PROGRAM EVACUAZIONE_SCARTI
VAR

	bINIT					:BOOL;
	
	//act Area MACINATORE
	rtAuto_ON				:R_TRIG;
	ftAuto_ON				:F_TRIG;
	tmrT3_ON				:TON;	
	tmrT3_OFF				:TON;		
	tmrT1T2_ON				:TON;	
	tmrT1T2_OFF				:TON;
	ft_AbilitaT1T2			:F_TRIG;
	ft_AbilitaT3			:F_TRIG;
	ft_AbilitaT4			:F_TRIG;
	
	Area_HS_On				:BOOL;
	rt_Area_M_Riarmo		:R_TRIG;
	rt_Area_M_Disarmo		:R_TRIG;
	tmr_SvuotaT1			:TON;		
	tmr_SvuotaT2			:TON;	
	tmr_SvuotaT3			:TON;	
	tmr_MacinatoreON		:TON;
	tmr_MacinatoreOFF		:TON;
	rt_MacinatoreON			:R_TRIG;
	rt_MacinatoreOFF		:R_TRIG;
	rt_MPO1_btn_M_MacOn		:R_TRIG;
	rt_btn_Fsx_T3StartMan	:R_TRIG;
	rt_btn_Fdx_T4StartMan	:R_TRIG;
	tmr_T3T5T6DelayStart	:TON;
	rt_T3S1full				:R_TRIG;
	tmr_T3S1vuoto			:TON;
	tmr_T3S1pieno			:TON;
	bT3S1full				:BOOL;
	rt_T3S2full				:R_TRIG;
	tmr_T3S2vuoto			:TON;
	bT3S2full				:BOOL;
	ft_T3S2full				:F_TRIG;
	countT3avanzamento		:INT;
	
	//act AREA SILOS
	rt_Area_S_Riarmo		:R_TRIG;
	rt_Area_S_Disarmo		:R_TRIG;
	
	//act_ALARM
	rtAlarmReset			:R_TRIG;	
	AlarmActive				:BOOL;
	AlarmReset				:BOOL;
	AlarmMask				:DWORD;
	T5_Bloccato				:ES_ALARM;	
	T6_Bloccato				:ES_ALARM;
	tmr_T4ON				:TON;
	
	tmrT3_Lavoro			:TON;	
	tmrT3_Pausa				:TON;
	tmrT5T6_RitStop			:TOF;	
	tmrS1_T_Rit_Empty		:TOF;
	tmrT1S01_Full			:TON;
	tmr_T_Rit_Stop_T4T5T6	:TOF;
	
	Forza_TT1S01_Full		:BOOL;
	
	appT1S01_Full			: BOOL;
	
	En_T_RitStopT5T6		:BOOL;
	
	//SENSORI	
	S1						:ES_S1;
	S2						:ES_S2;
	T1						:ES_T1;
	T3						:ES_T3;
	T5						:ES_T5;
	T6						:ES_T6;
                        	
	T1SO1tmravg				:TON;
	T1SO1arravg				:ARRAY[0..99]OF INT;
	T1SO1maxCnt				:INT;
	T1SO1sumavg				:REAL;
	T1SO1avg				:REAL;
	T1SO1cnt				:INT;
	T1SO1cnt2				:INT;	
	T1SO1cnt3				:INT;
	                    	
	S1SO2tmravg				:TON;
	S1SO2arravg				:ARRAY[0..99]OF INT;
	S1SO2maxCnt				:INT;
	S1SO2sumavg				:REAL;
	S1SO2avg				:REAL;
	S1SO2cnt				:INT;
	S1SO2cnt2				:INT;	
	S1SO2cnt3				:INT;		
                        	
	T3S1tmravg				:TON;
	T3S1arravg				:ARRAY[0..99]OF INT;
	T3S1maxCnt				:INT;
	T3S1sumavg				:REAL;
	T3S1avg					:REAL;
	T3S1cnt					:INT;
	T3S1cnt2				:INT;	
	T3S1cnt3				:INT;
	                    	
	T3S2tmravg				:TON;
	T3S2arravg				:ARRAY[0..99]OF INT;
	T3S2maxCnt				:INT;
	T3S2sumavg				:REAL;
	T3S2avg					:REAL;
	T3S2cnt					:INT;
	T3S2cnt2				:INT;	
	T3S2cnt3				:INT;
	                    	
	//SEMAFORI          	
	fbS1_Se1				:FB_Semaforo;
		
	//gestione filtro temporale sensore 
	SO2_full_curr			:BOOL;
	tmrValidaSoglia_S02		:TON;

	
	//gestione macinatore
	TON_Macinatore_On			:TON;
	TON_Vibro_Macinatore_On		:TON;
	TON_Ciclo_Macinatore		:TON;
	TP_Start_Macinatore			:TP;
	TP_Stop_Macinatore			:TP;

	TS							:BOOL;
	M_Ciclo_Svuotamento_Hdd_RUN	:BOOL;
	M_Auto_Start_Macinatore		:BOOL;
	M_Auto_Start_Vibro_Macinatore		:BOOL;
	M_Auto_Start_Vibro_Hdd		:BOOL;
	M_Start_Req_Stop_Macinatore	:BOOL;	
	M_Stop_Req_Stop_Macinatore	:BOOL;
	
	M_Man_Start_Vibro_Hdd		:BOOL;
	
	
	
	
	//TwinsAFE
	tmrErrAck				:TON;	
	
END_VAR
VAR // added by the converter: edge detectors and wires of the graphical bodies
    _rt1, _rt2 : R_TRIG;
    _w1, _w2, _w3 : BOOL;
    _ft1 : F_TRIG;
END_VAR


act_INIT();

act_ALARM();

act_INPUT();

act_Sensori();

act_AreaSilos();

act_Macinatore();

//act_AreaMac_AUTO();
//act_AreaMac_MAN();

act_Semafori();

act_OUTPUT();

act_HMI();

ACTION act_ALARM:

//TwinSAFE
TS_ErrAck := C1P1_Rst_Eme OR R1P1_Rst_Eme;


tmrErrAck(IN:=TS_ErrAck,PT:=T#1S);
IF tmrErrAck.Q THEN
	TS_ErrAck:=FALSE;
END_IF




//ALLARMI DA SENSORI
rtAlarmReset(CLK:=bAlarmReset);
IF rtAlarmReset.Q THEN
	bAlarmReset:=FALSE;
	T5.Alarm.Active:=FALSE;	
	T6.Alarm.Active:=FALSE;	
	bAllarmeT5:=FALSE;
	bAllarmeT6:=FALSE;
END_IF

IF NOT AlarmActive THEN

	//Allarme T5 Bloccato - 5s
	IF HQ1_T5_KA5 THEN
		T5.Alarm.tmr(IN:=TRUE,PT:=INT_TO_TIME(T5.Alarm.pt*1000));
		IF T5.Alarm.tmr.ET < T5.Alarm.tmr.PT THEN
			T5.S1_rt(CLK:=T5_S1);
			IF T5.S1_rt.Q THEN
				T5.S1_letto:=TRUE;		
			END_IF
		END_IF
	
		IF T5.Alarm.tmr.Q THEN
			IF NOT T5.S1_letto AND HQ1_T5_KA5 THEN
				T5.Alarm.Active:=TRUE AND bAllarmeT5enable;	
			ELSE	
				T5.Alarm.Active:=FALSE;	
			END_IF
			T5.S1_letto:=FALSE;
			T5.Alarm.tmr(IN:=FALSE);
		END_IF
	END_IF

	
	
		
	//Allarme T6 Bloccato - 5s
	IF HQ1_T6_KA6 THEN
		T6.Alarm.tmr(IN:=TRUE,PT:=INT_TO_TIME(T6.Alarm.pt*1000));
		IF T6.Alarm.tmr.ET < T6.Alarm.tmr.PT THEN
			T6.S1_rt(CLK:=T6_S1);
			IF T6.S1_rt.Q THEN
				T6.S1_letto:=TRUE;		
			END_IF
		END_IF
	
		IF T6.Alarm.tmr.Q THEN
			IF NOT T6.S1_letto AND HQ1_T6_KA6 THEN
				T6.Alarm.Active:=TRUE AND bAllarmeT6enable;	
			ELSE	
				T6.Alarm.Active:=FALSE;	
			END_IF
			T6.S1_letto:=FALSE;
			T6.Alarm.tmr(IN:=FALSE);
		END_IF	
	END_IF
	

	
	
	//Allarme S2 Silos Pieno
	IF S2.S1_full (*AND glo_ES_BtnHMI.S2_Alarm_Enable*) THEN
		S2.Alarm.Active := TRUE AND bAllarmeS2S1enable;
	END_IF
	
	
	
	
	//Allarme T3 Bloccato - 30s
	IF T1.SO1_full AND T3.S1_full THEN
		T3.Alarm.tmr(IN:=TRUE,PT:=INT_TO_TIME(T3.Alarm.pt*1000));
		IF T3.Alarm.tmr.Q THEN
			T3.Alarm.tmr(IN:=FALSE);
			T3.Alarm.Active := TRUE;	
		END_IF
	ELSE
		T3.Alarm.Active := FALSE;
	END_IF	

	
	
	
	//Allarme S1 Silos1 Pieno
	IF (*S1_S2_full AND*) S1_S2 THEN
		S1.Alarm.Active:=TRUE;
	END_IF
	
END_IF
END_ACTION

ACTION act_AreaMac_AUTO:

//#######################################################
//###################    AREA M ON    ###################
//#######################################################

IF M_PO1.key THEN
	rt_Area_M_Riarmo(CLK:= M_PO1.btn_R_Riarmo OR bSIMULA_btnR);
	IF rt_Area_M_Riarmo.Q THEN
		bSIMULA_btnR:=FALSE;
		AreaM_ON:= TRUE;
	END_IF
END_IF
rt_Area_M_Disarmo(CLK:= M_PO1.btn_0_AreaMoff OR bSIMULA_btn0);
IF NOT M_PO1.key OR rt_Area_M_Disarmo.Q OR NOT TS_AreaM_ON OR NOT TS_AreaS_ON (*OR NOT TS_AreaM_OFF*) THEN
	bSIMULA_btn0:=FALSE;	
	AreaM_ON:=FALSE;
	fun_AreaM_SPEGNITUTTO();	
END_IF

//#######################################################
//##################     AUTOMATICO   ###################
//#######################################################

rtAuto_ON(CLK:=HQ1_Auto_ON OR bSIMULAAuto_ON);
IF rtAuto_ON.Q THEN
	bIsAuto:=TRUE;
END_IF
ftAuto_ON(CLK:=HQ1_Auto_ON OR bSIMULAAuto_ON);
IF ftAuto_ON.Q THEN
	bIsAuto:=FALSE;	
	bSIMULA_btn0:=TRUE;	
	bSIMULA_btn0silos:=TRUE;	
	fun_AreaM_SPEGNITUTTO();	
END_IF

IF bIsAuto THEN
	

	//#######################################################
	//####################     T1 - T2    ###################
	//#######################################################
	
	(*
	- sensore sotto hundegger dà che T1 è pieno
	- area attiva
	- sensore all'inizio del T3 dà che è vuoto/libero
	- T3 non è bloccato: sensori del T1 e T3 contemporaneamente non pieni
	*)
	
	IF bAbilitaT1T2 THEN
		
		CASE stepT1T2 OF
			
			0:
				descT1T2:='T1-T2 spenti. In attesa di T1SO1 pieno';
				IF T1.SO1_full THEN
					stepT1T2:=5;
				END_IF
			
			5:
				IF NOT T3.S1_full (*AND NOT T3.Alarm.Active*) THEN 
					descT1T2:='Avvio T1-T2';
					bT1_ON:=TRUE;
					bT2_ON:=TRUE;
					tmrT1T2_ON(IN:=FALSE);
					stepT1T2:=10;
				ELSIF T3.S1_full (*OR T3.Alarm.Active*) THEN
					stepT1T2:=100;
				END_IF
			
			10:
				descT1T2:='T1-T2 accesi per 2s';
				tmrT1T2_ON(IN:=TRUE,PT:=T#2S);
				IF tmrT1T2_ON.Q THEN
					tmrT1T2_OFF(IN:=FALSE);
					stepT1T2:=15;					
				END_IF
			
			15:
				descT1T2:='T1-T2 accesi finchè T3S1 pieno';		
				IF NOT T1.SO1_full THEN
					tmrT1T2_ON(IN:=FALSE);					
					bT1_ON:=FALSE;
					stepT1T2:=16;
				END_IF		
				tmr_T3S1pieno(in:=T3.S1_full,PT:=T#2S);
				IF tmr_T3S1pieno.Q THEN
					bT1_ON:=FALSE;
					bT2_ON:=FALSE;
					stepT1T2:=20;				
				END_IF
	
			16:
				descT1T2:='T1spento, T2 acceso per 15s o finchè T3S1 pieno';	
				tmrT1T2_ON(IN:=TRUE,PT:=T#15S);	
				IF tmrT1T2_ON.Q OR T3.S1_full THEN
					bT2_ON:=FALSE;
					stepT1T2:=20;
				END_IF	
		
			20:
				descT1T2:='T1-T2 spenti, pausa 30s';
				tmrT1T2_OFF(IN:=TRUE,PT:=T#30S);
				IF tmrT1T2_OFF.Q THEN
					stepT1T2:=100;						
				END_IF
			
			100:
				tmrT1T2_OFF(IN:=FALSE);
				tmrT1T2_ON(IN:=FALSE);
				bT1_ON:=FALSE;
				bT2_ON:=FALSE;
				stepT1T2:=0;
					
		END_CASE
			
	END_IF
	ft_AbilitaT1T2(CLK:=bAbilitaT1T2);
	IF ft_AbilitaT1T2.Q THEN
		descT1T2:='T1-T2 disabilitati';
		HQ1_T1_KA1:=FALSE;
		HQ1_T2_KA2:=FALSE;
		bT1_ON:=FALSE;
		bT2_ON:=FALSE;
		stepT1T2:=100;			
	END_IF
	
	
	
	//#######################################################
	//##############    M - T3 - T5 - T6    #################
	//#######################################################
	
	(*
	- area attiva
	- bottone Macinatore da pulsantiera (vedi sotto fuori dall'automatico)
	- sensore all'inizio del T3 dà che è pieno
	- Silos2 non deve essere pieno
	- T5 non bloccato controllo paletta
	- T6 non bloccato controllo paletta
	*)
	IF NOT bAbilitaT3 THEN
		
		countT3avanzamento:=0;
		
	END_IF
	
	IF bAbilitaT3 THEN
	
		//azzeramento step automatici se il macinatore è stato avviato in locale
	//	IF NOT M_Start_Macinatore_Loc THEN
		//	stepT3 :=0;
	//	END_IF;
		CASE stepT3 OF
			
			0:
				descT3:='T3 fermo. In attesa di T3S1 pieno';
				IF NOT bT4_ON THEN// AND NOT M_Start_Macinatore_Loc THEN
					tmrT3_OFF(IN:=FALSE);
					tmrT3_ON(IN:=FALSE);
					IF T3.S1_full THEN	
						//PIENO INGRESSO, USCITA SCARICA -> ACCENDO T3						
						tT3ON_auto:=15;
						IF countT3avanzamento >=5 THEN
							descT3:='Macinatore acceso, attendo 20s per avvio T3';
							bM_ON:=TRUE;
							stepT3:=10;	
						ELSE
							descT3:='T3 acceso per 30s';
							bT3_ON:=TRUE;
							stepT3:=5;	
						END_IF	
					END_IF
				END_IF
		
			5:
				descT3:='T3 acceso per 30s';
				bT3_ON:=TRUE;
				tmrT3_ON(IN:=TRUE,PT:=INT_TO_TIME(tT3ON_auto*1000));
				IF tmrT3_ON.Q OR T3.S2_full THEN
					bT3_ON:=FALSE;	
					tmrT3_OFF(IN:=FALSE);
					countT3avanzamento:=countT3avanzamento+1;
					stepT3:=20;
				END_IF	
			
			10:
				descT3:='Macinatore acceso, attendo 20s per avvio T3';
				tmrT3_OFF(IN:=TRUE,PT:=T#20S);
				IF tmrT3_OFF.Q THEN
					bT3_ON:=TRUE;
					T3_ModoPausaLavoro:=TRUE;
					bT3EnT1PausaLavoro:=TRUE;  (*abilito un timer per far lavorare T3 pausa-lavoro per non intasare T5*)
					bT3EnT2PausaLavoro:=FALSE;
					T3_Lavoro:=TRUE;
					stepT3:=15;
				END_IF
		
			15:
				descT3:='T3 e Macinatore accesi per 5min';
				tmrT3_ON(IN:=TRUE,PT:=T#8M);
				IF tmrT3_ON.Q THEN
					tmrT3_OFF(IN:=FALSE);
					bM_ON:=FALSE;
					bT3_ON:=FALSE;
					T3_ModoPausaLavoro:=FALSE;
					bT3EnT1PausaLavoro:=FALSE;
					bT3EnT2PausaLavoro:=FALSE;
					T3_Lavoro:=FALSE;
					stepT3:=20;
					countT3avanzamento:=0;
				END_IF
				
			20:
				descT3:='Tutto spento, pausa di 30s';
				tmrT3_OFF(IN:=TRUE,PT:=T#30S);
				IF tmrT3_OFF.Q THEN
					tmrT3_OFF(IN:=FALSE);
					stepT3:=0;
				END_IF
			
			100:
				tmrT3_OFF(IN:=FALSE);
				tmrT3_ON(IN:=FALSE);
				bM_ON:=FALSE;
				stepT3:=0;
		
		END_CASE
	
	END_IF
	ft_AbilitaT3(CLK:=bAbilitaT3);
	IF ft_AbilitaT3.Q THEN
		descT3:='T3 disabilitato';
		HQ1_T3_KA3:=FALSE;	
		bMacinatoreStart:=FALSE;
		bMacinatoreStop:=TRUE;
		stepT3:=100;		
	END_IF
	
	
	
	//#######################################################
	//#################     T4 - T5 - T6    #################
	//#######################################################
	
	(*
	- T5 non bloccato controllo paletta
	- T6 non bloccato controllo paletta
	- Silos2 non deve essere pieno
	- Consenso da logica Aspirazione
	*)
	
	IF bAbilitaT4 THEN
		
		CASE stepT4 OF
			
		0:
			descT4:='T4 fermo. In attesa di LogicaAspirazioneON';
			IF (NOT bT3_ON AND bMacinatoreStop) AND LogicaAspirazioneON THEN
				bT4_ON:=TRUE;
				stepT4:=10;
			END_IF
		
		10:
			descT4:='T4 acceso per 30s';
			tmr_T4ON(IN:=TRUE,PT:=T#30S);	
			IF tmr_T4ON.Q THEN
				tmr_T4ON(IN:=FALSE);
				IF NOT LogicaAspirazioneON THEN
					stepT4:=100;			
				END_IF				
			END_IF
			
		100:
			tmr_T4ON(IN:=FALSE);
			bT4_ON:=FALSE;
			stepT4:=0;
					
		END_CASE

	END_IF
	ft_AbilitaT4(CLK:=bAbilitaT4);
	IF ft_AbilitaT4.Q THEN
		descT4:='T4 disabilitato';
		HQ1_T4_KA4:=FALSE;
		bT4_ON:=FALSE;
		stepT4:=100;			
	END_IF
	
END_IF



//####################################################################
//####     GESTIONE TIMER PAUSA LAVORO IN CICLO AUTOMATICO T3 #######
//###################################################################

tmrT3_Lavoro(IN:=bT3EnT1PausaLavoro,PT:=T#20S);
tmrT3_Pausa(IN:=bT3EnT2PausaLavoro,PT:=T#30S);

IF tmrT3_Lavoro.Q THEN
	bT3EnT1PausaLavoro := FALSE;	
	bT3EnT2PausaLavoro := TRUE;
	T3_Lavoro := FALSE;	
END_IF

IF tmrT3_Pausa.Q THEN
	bT3EnT1PausaLavoro := TRUE;	
	bT3EnT2PausaLavoro := FALSE;
	T3_Lavoro := TRUE;
END_IF

//##################################################################
//####     		 GESTIONE TIMER RITARDO STOP T5-T6	 		 #######
//##################################################################
En_T_RitStopT5T6 := bM_ON AND AreaM_ON;
tmrT5T6_RitStop(IN:=En_T_RitStopT5T6,PT:=T#30S);

//#######################################################
//####     USCITE INDIPENDENDI DA MODO AUTO/MAN   #######
//#######################################################

HQ1_T1_KA1:= bT1_ON AND AreaM_ON;
HQ1_T2_KA2:= bT2_ON AND AreaM_ON;

M_Cmd_T3 := bT3_ON AND (T3_Lavoro OR NOT T3_ModoPausaLavoro);

HQ1_T3_KA3:= M_Cmd_T3 AND NOT SensInMac AND AreaM_ON AND NOT (T5.Alarm.Active OR T6.Alarm.Active OR S2.Alarm.Active);		
HQ1_T4_KA4:= bT4_ON AND AreaM_ON AND LogicaAspirazioneON AND NOT (T5.Alarm.Active OR T6.Alarm.Active OR S2.Alarm.Active);
HQ1_T5_KA5:= (bM_ON OR bT4_ON OR tmrT5T6_RitStop.Q) AND AreaM_ON AND NOT (T5.Alarm.Active OR T6.Alarm.Active OR S2.Alarm.Active);
HQ1_T6_KA6:= (bM_ON OR bT4_ON OR tmrT5T6_RitStop.Q) AND AreaM_ON AND NOT T6.Alarm.Active AND NOT S2.Alarm.Active;
		

bMacinatoreStart:= bM_ON AND AreaM_ON AND NOT (T5.Alarm.Active AND T6.Alarm.Active AND S2.Alarm.Active) and HQ1_T5_KA5;
bMacinatoreStop:= NOT bM_ON OR T5.Alarm.Active OR T6.Alarm.Active OR NOT HQ1_T5_KA5 OR NOT HQ1_T5_KA5;	

//#######################################################
//#############     START-STOP MACINATORE   #############
//#######################################################

//AVVIO MACINATORE RICHIEDE CHE DOPO 1s USCITA VENGA ABBASSATA
rt_MacinatoreON(CLK:=bMacinatoreStart);	
IF rt_MacinatoreON.Q THEN
	HQ1_M_ON:=TRUE;
	HQ1_M_OFF:=FALSE;

END_IF
tmr_MacinatoreON(IN:=HQ1_M_ON,PT:=T#1S);	
IF tmr_MacinatoreON.Q THEN
	tmr_MacinatoreON(IN:=FALSE);
	HQ1_M_ON:=FALSE;
END_IF
//SPEGNIMENTO MACINATORE RICHIEDE CHE DOPO 1s USCITA VENGA ABBASSATA
rt_MacinatoreOFF(CLK:=bMacinatoreStop);	
IF rt_MacinatoreOFF.Q THEN
	HQ1_M_ON:=FALSE;
	HQ1_M_OFF:=TRUE;

END_IF
tmr_MacinatoreOFF(IN:=HQ1_M_OFF,PT:=T#1S);	
IF tmr_MacinatoreOFF.Q THEN
	tmr_MacinatoreOFF(IN:=FALSE);
	HQ1_M_OFF:=FALSE;
END_IF
	
		
	
	

//#######################################################
//##################     PULSANTIERA   ##################
//#######################################################

IF AreaM_ON AND bAbilitaPulsatiera THEN
	
	//M	
	rt_MPO1_btn_M_MacOn(CLK:=(M_PO1.btn_M_MacOn OR bSIMULA_btnM));
	IF rt_MPO1_btn_M_MacOn.Q AND bMacinatoreStop THEN
		bSIMULA_btnM:=FALSE;
		//M SPENTO -> LO ACCENDO
		bM_ON:=TRUE;
		IF NOT SensInMac AND NOT HQ1_T4_KA4 THEN
			bT3T5T6DelayStart:= TRUE;
		END_IF		
	ELSIF rt_MPO1_btn_M_MacOn.Q AND bMacinatoreStart THEN
		//M ACCESO -> LO SPENGO
		bSIMULA_btnM:=FALSE;
		bM_ON:=FALSE;	
		bT3T5T6DelayStart:=FALSE;
		IF (*NOT M_PO1.btn_Fsx_T3StartMan AND*) NOT glo_ES_ActVal.PuliziaT1t2_ON THEN
			bT3_ON:=FALSE;
			M_Start_Macinatore_Loc := FALSE;
		END_IF
	END_IF
	
	IF (T5.Alarm.Active OR T6.Alarm.Active OR S2.Alarm.Active) THEN
		bM_ON:=FALSE;
	END_IF
		
	//AVVIO RITARDATO DEL T3,T5,T6 DOPO 15s DALL'AVVIO M	
	tmr_T3T5T6DelayStart(IN:=bT3T5T6DelayStart, PT:=T#35S);
	IF tmr_T3T5T6DelayStart.Q THEN
		bT3T5T6DelayStart:=FALSE;
		bT3_ON:=TRUE;
		M_Start_Macinatore_Loc := TRUE;
	END_IF
	
	//T3
	rt_btn_Fsx_T3StartMan(CLK:=M_PO1.btn_Fsx_T3StartMan OR bSIMULA_btnT3);		//FRECCIA A SINISTRA SU BOTTONE DI SINISTRA
	IF rt_btn_Fsx_T3StartMan.Q THEN
		IF NOT SensInMac AND NOT HQ1_T3_KA3 THEN				//SE SENSORE SU MAC è ON, ALLORA NN ACCENDO T3 XKE LO INTASO
			bSIMULA_btnT3:=FALSE;
			bT3_ON:= TRUE;
		ELSIF NOT glo_ES_ActVal.PuliziaT1t2_ON AND HQ1_T3_KA3 THEN
			bSIMULA_btnT3:=FALSE;
			bT3_ON:=FALSE;
		END_IF			
	END_IF
	
	IF NOT bM_ON THEN 
		bT3_ON:=FALSE;
	END_IF
	
	//T4
	rt_btn_Fdx_T4StartMan(CLK:=M_PO1.btn_Fsx_T4StartMan);
	IF rt_btn_Fdx_T4StartMan.Q THEN		//FRECCIA A SINISTRA SU BOTTONE DI DESTRA
		IF NOT HQ1_T4_KA4 THEN	
			bT4_ON:= TRUE;
		ELSE
			bT4_ON:=FALSE;
		END_IF
	END_IF
		
	//T7
	IF M_PO1.btn_Fup_T7Avanti THEN			//FRECCIA IN SU
		HQ1_T7_A_KA8:= TRUE;
		HQ1_T7_I_KA9:= FALSE;
	ELSIF M_PO1.btn_Fdw_T7Indietro THEN		//FRECCIA IN GIU'
		HQ1_T7_I_KA9:= TRUE;
		HQ1_T7_A_KA8:=FALSE;
	ELSE
		HQ1_T7_A_KA8:=FALSE;
		HQ1_T7_I_KA9:= FALSE;
	END_IF
	
END_IF
END_ACTION

ACTION act_AreaMac_MAN:

//#######################################################
//####################     MANUALE   ####################
//#######################################################


IF NOT bIsAuto THEN
		
	//#######################################################
	//###############     PULIZIA T1-T2-T3   ################
	//#######################################################

	IF 	bMAN_SvuotaT1T2T3 THEN
		bMAN_SvuotaT1T2T3:=FALSE;
		glo_ES_ActVal.PuliziaT1T2_ON:=TRUE;
		bT1_ON:= TRUE;
		bT2_ON:= TRUE;
		bM_ON:= TRUE;
		bT3T5T6DelayStart:=TRUE;
	END_IF
	IF glo_ES_ActVal.PuliziaT1T2_ON THEN
		tmr_SvuotaT1(IN:= bT1_ON,PT:=DINT_TO_TIME(glo_ES_Config.T1_Time*1000));
		tmr_SvuotaT2(IN:= bT2_ON,PT:=DINT_TO_TIME(glo_ES_Config.T2_Time*1000));
		tmr_SvuotaT3(IN:= bM_ON,PT:=DINT_TO_TIME(glo_ES_Config.T3_Time*1000));
	END_IF

	//STOP T1
	IF tmr_SvuotaT1.Q THEN
		tmr_SvuotaT1(IN:=FALSE);
		bT1_ON:= FALSE;
	END_IF
		
	//STOP T2
	IF tmr_SvuotaT2.Q THEN
		tmr_SvuotaT2(IN:=FALSE);
		bT2_ON:= FALSE;
	END_IF
	
	//STOP T3	
	IF tmr_SvuotaT3.Q THEN
		tmr_SvuotaT3(IN:=FALSE);
		bM_ON:= FALSE;
		bT3T5T6DelayStart:=FALSE;
		glo_ES_ActVal.PuliziaT1t2_ON:=FALSE;
	END_IF

	
	//#######################################################
	//#################     PULIZIA S1-T4   #################
	//#######################################################
	
	IF bMAN_SvuotaS1T4 THEN
		bMAN_SvuotaS1T4:=FALSE;
		
	END_IF
	
	
END_IF
END_ACTION

ACTION act_AreaSilos:

//#######################################################
//###################    AREA S ON    ###################
//#######################################################

IF S1_PO1.key THEN
	rt_Area_S_Riarmo(CLK:= S1_PO1.btn_R_Riarmo OR bSIMULA_btnRsilos);
	IF rt_Area_S_Riarmo.Q THEN
		bSIMULA_btnRsilos:=FALSE;
		AreaS_ON:= TRUE;
	END_IF
END_IF
rt_Area_S_Disarmo(CLK:= S1_PO1.btn_0_AreaMoff OR bSIMULA_btn0silos);
IF NOT S1_PO1.key OR rt_Area_S_Disarmo.Q OR NOT TS_AreaM_ON OR NOT TS_AreaS_ON (*OR TS_AreaS_OFF*) THEN
	bSIMULA_btn0silos:=FALSE;	
	AreaS_ON:=FALSE;
END_IF

	//led pulsante area macinatore ON
	S1_PO1.led_0_AreaMoff := AreaS_ON;

	//led pulsante riarmo area macinatore
	S1_PO1.led_R_Riarmo := TS_AreaS_ON;
	
	//riarmo emergenze
//	TS_S1PO1_btn_R := S1_PO1.key AND S1_PO1.btn_R_Riarmo;
	TS_S1PO1_btn_R := S1_PO1.key AND(C1P1_Rst_Eme OR R1P1_Rst_Eme);
	
	
//#######################################################
//#############    LOGICA M-ASPIRAZIONE   ###############
//#######################################################

IF AreaS_ON AND bAbilitaPulsatieraS1PO1 THEN
	
	//VALVOLA STELLARE S1_SO2	
	IF (S1.SO2_full) AND NOT bT3_ON AND bMacinatoreStop AND NOT bSIMULA_BrichettatriceON AND bAbilitaT4 THEN
		HQ1_S1_ValvolaStellare:=TRUE;
	ELSE
		HQ1_S1_ValvolaStellare:=FALSE;
	END_IF
	
//	HQ1_S1_ValvolaStellare:=FALSE;
	
	//BRICCHETTATRICE
	IF (*HQ1_ScorniciatriceON AND NOT HQ1_S1_ValvolaStellare AND*) bSIMULA_BrichettatriceON THEN
		HQ1_BrichettatriceON:=TRUE;
	ELSE
		HQ1_BrichettatriceON:=FALSE;
	END_IF
	
	//RACLA
	IF HQ1_BrichettatriceON OR HQ1_S1_ValvolaStellare THEN
		HQ1_RaclaON:=TRUE;
	ELSE
		HQ1_RaclaON:=FALSE;
	END_IF 
	
	//CONSENSO A T4 T5 T6
tmr_T_Rit_Stop_T4T5T6(IN:=HQ1_S1_ValvolaStellare,PT:=T#1M);
	
IF tmr_T_Rit_Stop_T4T5T6.Q THEN
		LogicaAspirazioneON:=TRUE;
	ELSE
		LogicaAspirazioneON:=FALSE;		
	END_IF
	
END_IF
END_ACTION

ACTION act_HMI:


bAllarmeT3	:= T3.Alarm.Active;			
bAllarmeT5	:= T5.Alarm.Active;			
bAllarmeT6	:= T6.Alarm.Active;
bAllarmeS2S1:= S2.Alarm.Active;

bT1SO1pieno	:= T1.SO1_full;
bT3S1pieno	:= T3.S1_full;
bT3S2pieno	:= T3.S2_full;
bS1SO2pieno	:= S1.SO2_full;
bS2S1pieno	:= S2.S1_full;

glo_ES_ActVal.T3_S1:= T3.S1_actVal;
glo_ES_ActVal.T3_S2:= T3.S2_actVal;
glo_ES_ActVal.S2_S1:= S2.S1_actVal;
glo_ES_ActVal_T1_SO1:= T1_SO1;

altMatT3S1:=T3.S1_fb.distanzaAVuoto - T3.S1_actVal;
IF altMatT3S1 <0 THEN
	altMatT3S1:=0;
END_IF
altMatT3S2:=T3.S2_fb.distanzaAVuoto - T3.S2_actVal;
IF altMatT3S2 <0 THEN
	altMatT3S2:=0;
END_IF 
distMatT1SO1:= T1.SO1_fb.distanzaAVuoto - T1.SO1_actVal;
IF distMatT1SO1 <0 THEN
	distMatT1SO1:=0;
END_IF 

IF sogliaT3S1 = 0 THEN
	sogliaT3S1:=100;
END_IF
IF sogliaT3S2 = 0 THEN
	sogliaT3S2:=40;
END_IF
//IF sogliaS1SO2 = 0 THEN
//	sogliaS1SO2:=1000;
//END_IF
IF solgiaT1SO1 = 0 THEN
	solgiaT1SO1:=5000;
END_IF
END_ACTION

ACTION act_INIT:

IF NOT bINIT THEN
	
	bINIT:=TRUE;

	bMacinatoreStop:=TRUE;

	//Avvia TwinSAFE Gruppo EVACUAZIONE SCARTI
	TS_Run_GrpES:=TRUE;

END_IF
END_ACTION

ACTION act_INPUT:

//TERM7 EL1008 H-Q1
SensInMac				:= glo_dig_in_HQ1[1];		//DIGIN CH1			Sensore ingresso macinatore
R5_S2					:= glo_dig_in_HQ1[2];		//DIGIN CH2			Val1 aperta
T5_S3					:= glo_dig_in_HQ1[3];		//DIGIN CH3			Val2 chiusa
S1_S3					:= glo_dig_in_HQ1[4];		//DIGIN CH4			Allarme silos1 pieno
T6_S1					:= glo_dig_in_HQ1[5];		//DIGIN CH5			Rotaz catena IFS289
HQ1_Auto_ON				:= glo_dig_in_HQ1[6];		//DIGIN CH6			Modo auto-man
HQ1_P1					:= glo_dig_in_HQ1[7];		//DIGIN CH7			Reset Allarme
HQ1_K1					:= glo_dig_in_HQ1[8];		//DIGIN CH8			---

//TERM8 EL1008 H-Q1
//HQ1_AspirazioneON		:= glo_dig_in_HQ1[10];		//DIGIN CH2			Motore aspirazione in silos S1
I_Fdbk_Km_Area_Nastri_Macinatore:= glo_dig_in_HQ1[9];		//DIGIN CH2			feedback contattore area macinatore
I_Fdbk_Km_Area_Macinatore:= glo_dig_in_HQ1[10];		//DIGIN CH2			feedback contattore area macinatore
I_Macinatore_Run		:= glo_dig_in_HQ1[12];		//DIGIN CH1			Scorniciatrice accesa

S1_S2					:= glo_dig_in_HQ1[12];		//DIGIN CH4			Sensore troppopieno in alto in silos S1
S1_S1					:= glo_dig_in_HQ1[13];		//DIGIN CH5			Sensore livello in basso in silos S1
HQ1_BricchettatriceON	:= glo_dig_in_HQ1[13];		//DIGIN CH6			Bricchettatrice accesa



//TERM11 EL3012 H-Q1
T3_S1					:= glo_analog_in_HQ1[1];	//ANALOGIN CH1		Pres materiale In T3
T3_S2					:= glo_analog_in_HQ1[2];	//ANALOGIN CH2		Pres materiale Out T3

//TERM12 EL3012 H-Q1
S1_SO2					:= glo_analog_in_HQ1[3];	//ANALOGIN CH1		Liv silos2 UMT 30-6000


(*****************************************************************)	
(*****************************************************************)	
(*****************************************************************)

//BOX16 EP6228-0022 M-CS1
T1_SO1					:= glo_analog_in_MCS1[1];	//IOLINK CH1	Già in mm. Pres mat T1, da inizio vibro fino sopra nastro  O1D120


(*****************************************************************)	
(*****************************************************************)	
(*****************************************************************)

//BOX17 EP6228-0022 T3-C01
S2_S1					:= glo_analog_in_T3C01[1];	//IOLINK CH2		LIV AVVIO VALV STELLARE UGT514

//S1_PO1											//IOLINK CH3		PULSANTIERA BNI005N
S1_PO1.key				:= glo_dig_in_T3C01[1];		//CHIAVE
S1_PO1.btn_0_AreaMoff	:= glo_dig_in_T3C01[2];		//BOTTONE '0'
S1_PO1.btn_R_Riarmo		:= glo_dig_in_T3C01[3];		//BOTTONE 'r'
I_Pls_Start_Vibro_Hdd	:= glo_dig_in_T3C01[7];

//M_PO1												//IOLINK CH4		PULSANTIERA BNI005M
M_PO1.key				:= glo_dig_in_T3C01[1];		//CHIAVE
M_PO1.btn_0_AreaMoff	:= glo_dig_in_T3C01[2];	//BOTTONE '0'
M_PO1.btn_R_Riarmo		:= glo_dig_in_T3C01[3];	//BOTTONE 'r'
M_PO1.btn_M_MacOn		:= glo_dig_in_T3C01[4];	//TASTO 'M'
M_PO1.btn_Fdw_T7Indietro:= glo_dig_in_T3C01[13];	//FRECCIA IN GIU'
M_PO1.btn_Fup_T7Avanti	:= glo_dig_in_T3C01[14];	//FRECCIA IN SU
M_PO1.btn_Fsx_T3StartMan:= glo_dig_in_T3C01[15];	//FRECCIA SX BTN SX
M_PO1.btn_Fsx_T4StartMan:= glo_dig_in_T3C01[16];	//FRECCIA SX BTN DX

T5_S1					:= glo_dig_in_T3C01[25];	//DIGIN  CH7		ROTAZ CATENA IFS289
T5_SO1					:= glo_analog_in_T3C01[2];	//IOLINK CH8		LIV SCARICO MAC UGT525

//
I_Barriera_Macinatore := glo_dig_in_T3C01[10];
END_ACTION

ACTION act_Macinatore:
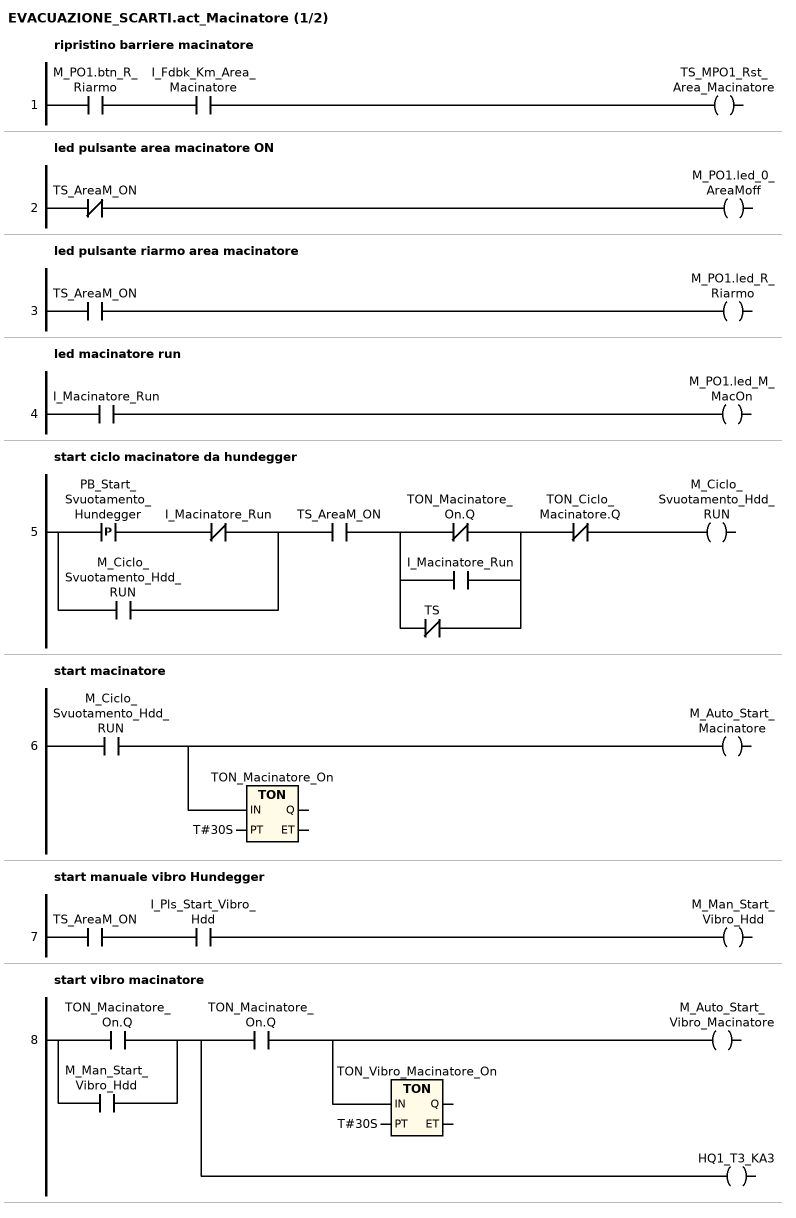
// NETWORK 1: ripristino barriere macinatore
TS_MPO1_Rst_Area_Macinatore := M_PO1.btn_R_Riarmo AND I_Fdbk_Km_Area_Macinatore;

// NETWORK 2: led pulsante area macinatore ON
M_PO1.led_0_AreaMoff := NOT TS_AreaM_ON;

// NETWORK 3: led pulsante riarmo area macinatore
M_PO1.led_R_Riarmo := TS_AreaM_ON;

// NETWORK 4: led macinatore run
M_PO1.led_M_MacOn := I_Macinatore_Run;

// NETWORK 5: start ciclo macinatore da hundegger
_rt1(CLK := PB_Start_Svuotamento_Hundegger);
M_Ciclo_Svuotamento_Hdd_RUN := (_rt1.Q AND NOT I_Macinatore_Run OR M_Ciclo_Svuotamento_Hdd_RUN) AND TS_AreaM_ON AND (NOT TON_Macinatore_On.Q OR I_Macinatore_Run OR NOT TS) AND NOT TON_Ciclo_Macinatore.Q;

// NETWORK 6: start macinatore
M_Auto_Start_Macinatore := M_Ciclo_Svuotamento_Hdd_RUN;
TON_Macinatore_On(IN := M_Ciclo_Svuotamento_Hdd_RUN, PT := T#30S); // TON

// NETWORK 7: start manuale vibro Hundegger
M_Man_Start_Vibro_Hdd := TS_AreaM_ON AND I_Pls_Start_Vibro_Hdd;

// NETWORK 8: start vibro macinatore
_w1 := TON_Macinatore_On.Q OR M_Man_Start_Vibro_Hdd;
_w2 := _w1 AND TON_Macinatore_On.Q;
M_Auto_Start_Vibro_Macinatore := _w2;
TON_Vibro_Macinatore_On(IN := _w2, PT := T#30S); // TON
HQ1_T3_KA3 := _w1;

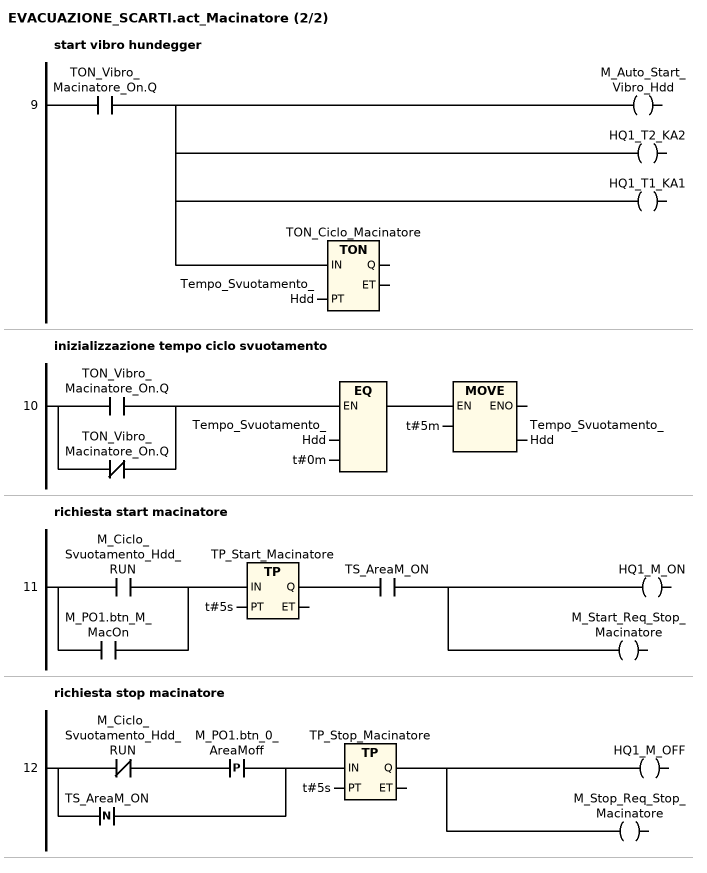
// NETWORK 9: start vibro hundegger
M_Auto_Start_Vibro_Hdd := TON_Vibro_Macinatore_On.Q;
HQ1_T2_KA2 := TON_Vibro_Macinatore_On.Q;
HQ1_T1_KA1 := TON_Vibro_Macinatore_On.Q;
TON_Ciclo_Macinatore(IN := TON_Vibro_Macinatore_On.Q, PT := Tempo_Svuotamento_Hdd); // TON

// NETWORK 10: inizializzazione tempo ciclo svuotamento
IF (TON_Vibro_Macinatore_On.Q OR NOT TON_Vibro_Macinatore_On.Q) AND Tempo_Svuotamento_Hdd = t#0m THEN
    Tempo_Svuotamento_Hdd := t#5m;
END_IF

// NETWORK 11: richiesta start macinatore
TP_Start_Macinatore(IN := M_Ciclo_Svuotamento_Hdd_RUN OR M_PO1.btn_M_MacOn, PT := t#5s); // TP
_w3 := TP_Start_Macinatore.Q AND TS_AreaM_ON;
HQ1_M_ON := _w3;
M_Start_Req_Stop_Macinatore := _w3;

// NETWORK 12: richiesta stop macinatore
_rt2(CLK := M_PO1.btn_0_AreaMoff);
_ft1(CLK := TS_AreaM_ON);
TP_Stop_Macinatore(IN := NOT M_Ciclo_Svuotamento_Hdd_RUN AND _rt2.Q OR _ft1.Q, PT := t#5s); // TP
HQ1_M_OFF := TP_Stop_Macinatore.Q;
M_Stop_Req_Stop_Macinatore := TP_Stop_Macinatore.Q;
END_ACTION

ACTION act_OUTPUT:

IF NOT bSIMULA_out THEN
	
	//TERM9 EL2008 H-Q1
	glo_dig_out_HQ1[1]		:=	Dis_Scarico_Hundegger;//S1_U1;									//DIGOUT CH1		Valvola aria pulizia ingresso M12
	glo_dig_out_HQ1[2]		:=	HQ1_T1_KA1;								//DIGOUT CH2		T1 Vibrotrasp buca
	glo_dig_out_HQ1[3]		:=	HQ1_T2_KA2;								//DIGOUT CH3		T2 Nastro elev buca
	glo_dig_out_HQ1[4]		:=	HQ1_T3_KA3;// AND NOT SensInMac;			//DIGOUT CH4		T3 Vibrotrasp macinatore
	glo_dig_out_HQ1[5]		:=	HQ1_T5M2_A_KA4;							//DIGOUT CH5		Apre scarico trasp orizz
	glo_dig_out_HQ1[6]		:=	HQ1_T5_KA5;								//DIGOUT CH6		Trasp elevat a parete
	glo_dig_out_HQ1[7]		:=	HQ1_T6_KA6;								//DIGOUT CH7		Trasp orizza a parete
	glo_dig_out_HQ1[8]		:=	HQ1_T5M2_C_KA7;							//DIGOUT CH8		Chiude scarico trasp orizz
	
	//TERM10 EL2008 H-Q1
	glo_dig_out_HQ1[9]		:= HQ1_T7_A_KA8;							//DIGOUT CH1		Caricatore macinat Avanti
	glo_dig_out_HQ1[10]		:= HQ1_T7_I_KA9;							//DIGOUT CH2		Caricatore macinat Indietro
	glo_dig_out_HQ1[11]		:= HQ1_M_ON;								//DIGOUT CH3		Macinatore ON impulsivo
	glo_dig_out_HQ1[12]		:= HQ1_M_OFF;								//DIGOUT CH4		Macinatore OFF impulsivo
	glo_dig_out_HQ1[13]		:= HQ1_T4_KA4;								//DIGOUT CH5		T4 Trasportatore silos macinatore	
	glo_dig_out_HQ1[14]		:= HQ1_S1_ValvolaStellare;					//DIGOUT CH6		Valvola stellare scarico silos 1	
	glo_dig_out_HQ1[15]		:= HQ1_RaclaON;								//DIGOUT CH7		Rancia: avviata da quadro silos
	glo_dig_out_HQ1[16]		:= HQ1_BrichettatriceON;					//DIGOUT CH8		Bricchettatrice: avviata da quadro silos

	//M_PO1											
	//IOLINK CH4		PULSANTIERA BNI005M
	glo_dig_out_T3C01[5] 	:= M_PO1.led_M_MacOn;						//BOTTONE '0'
	glo_dig_out_T3C01[8]	:= M_PO1.led_R_Riarmo;						//BOTTONE 'r'
	glo_dig_out_T3C01[6]	:= M_PO1.led_0_AreaMoff;					//TASTO 'M'
	
	//S1_PO1											
	//IOLINK CH4		PULSANTIERA BNI005M
					//BOTTONE 'r'

END_IF
END_ACTION

ACTION act_Semafori:

//#######################################################
//####################    SEMAFORI   ####################
//#######################################################

IF TS_AreaM_ON THEN
	IF I_Macinatore_Run  THEN
		fbS1_Se1(bON:= TRUE, sColore:= 3, bBlink:= TRUE, semaforo=> S1_Se1);	//verde	
	ELSE
		fbS1_Se1(bON:= TRUE, sColore:= 4, bBlink:= TRUE, semaforo=> S1_Se1);	//arancio
	END_IF
ELSE	
	fbS1_Se1(bON:= TRUE, sColore:= 2, bBlink:= TRUE, semaforo=> S1_Se1);	//rosso
END_IF
END_ACTION

ACTION act_Sensori:

//#######################################################
//####################    SENSORI   #####################
//#######################################################
//SOTTO HUNDEGGER
//CODA CIRCOLARE VALORI SENSORE inbit
T1SO1tmravg(IN:=TRUE,PT:=T#200MS);
T1SO1maxCnt:= REAL_TO_INT(T1SO1maxTimeavg*1000/200);
IF T1SO1maxCnt > 99 THEN
	T1SO1maxCnt:=99;
END_IF
IF T1SO1tmravg.Q THEN
	T1SO1tmravg(IN:=FALSE);	
	//CONTATORE TEMPO MASSIMO CAMPIONATURA
	IF T1SO1cnt < T1SO1maxCnt-1 THEN
		T1SO1cnt:=T1SO1cnt+1;	
	ELSE
		T1SO1cnt:=0;
	END_IF
	//POPOLO ARRAY LETTURE SENSORE in bit			
	T1SO1arravg[T1SO1cnt]:= T1_SO1;
END_IF
//MEDIA VALORI inbit
T1SO1cnt3:=0;
T1SO1sumavg:=0;
FOR T1SO1cnt2:=1 TO T1SO1maxCnt-1 DO
	IF T1SO1arravg[T1SO1cnt2] > 0 THEN
		T1SO1sumavg:= T1SO1sumavg + T1SO1arravg[T1SO1cnt2];
		T1SO1cnt3:=T1SO1cnt3+1;
	END_IF
END_FOR
IF T1SO1sumavg > 0 THEN
	T1SO1avg:=(T1SO1sumavg/T1SO1cnt3);	
END_IF
T1.SO1_fb(
	lettura:= REAL_TO_INT(T1SO1avg), 
	distanzaAVuoto:=6150,
	valSoglia:= solgiaT1SO1, 
	filtertime:=0,
	full=> appT1S01_Full);		
	
	//T1S01 full ritardato di 10 secondi 
	tmrT1S01_Full(IN:=appT1S01_Full,PT:=T#10S);
	T1.SO1_full := tmrT1S01_Full.Q;
	
//INGRESSO al T3
//CODA CIRCOLARE VALORI SENSORE inbit
T3S1tmravg(IN:=TRUE,PT:=T#200MS);
T3S1maxCnt:= REAL_TO_INT(T3S1maxTimeavg*1000/200);
IF T3S1maxCnt > 99 THEN
	T3S1maxCnt:=99;
END_IF
IF T3S1tmravg.Q THEN
	T3S1tmravg(IN:=FALSE);	
	//CONTATORE TEMPO MASSIMO CAMPIONATURA
	IF T3S1cnt < T3S1maxCnt-1 THEN
		T3S1cnt:=T3S1cnt+1;	
	ELSE
		T3S1cnt:=0;
	END_IF
	//POPOLO ARRAY LETTURE SENSORE in bit			
	T3S1arravg[T3S1cnt]:= T3_S1;
END_IF
//MEDIA VALORI inbit
T3S1cnt3:=0;
T3S1sumavg:=0;
FOR T3S1cnt2:=1 TO T3S1maxCnt-1 DO
	IF T3S1arravg[T3S1cnt2] > 0 THEN
		T3S1sumavg:= T3S1sumavg + T3S1arravg[T3S1cnt2];
		T3S1cnt3:=T3S1cnt3+1;
	END_IF
END_FOR
IF T3S1sumavg > 0 THEN
	T3S1avg:=(T3S1sumavg/T3S1cnt3);	
END_IF
T3.S1_fb(
	lettura:= REAL_TO_INT(T3S1avg), 
	maxScaleBit:= 32767, 
	maxScaleIng:= 1300, 
	deltaLowLimit:= 30,
	distanzaAVuoto:=1173,
	valSoglia:= sogliaT3S1, 
	filterTime:=2,
	full=> T3.S1_full,
	actualVal=> T3.S1_actVal);


//USCITA al T3	
//CODA CIRCOLARE VALORI SENSORE inbit
T3S2tmravg(IN:=TRUE,PT:=T#200MS);
T3S2maxCnt:= REAL_TO_INT(T3S2maxTimeavg*1000/200);
IF T3S2maxCnt > 99 THEN
	T3S2maxCnt:=99;
END_IF
IF T3S2tmravg.Q THEN
	T3S2tmravg(IN:=FALSE);	
	//CONTATORE TEMPO MASSIMO CAMPIONATURA
	IF T3S2cnt < T3S2maxCnt-1 THEN
		T3S2cnt:=T3S2cnt+1;	
	ELSE
		T3S2cnt:=0;
	END_IF
	//POPOLO ARRAY LETTURE SENSORE in bit			
	T3S2arravg[T3S2cnt]:= T3_S2;
END_IF
//MEDIA VALORI inbit
T3S2cnt3:=0;
T3S2sumavg:=0;
FOR T3S2cnt2:=1 TO T3S2maxCnt-1 DO
	IF T3S2arravg[T3S2cnt2] > 0 THEN
		T3S2sumavg:= T3S2sumavg + T3S2arravg[T3S2cnt2];
		T3S2cnt3:=T3S2cnt3+1;
	END_IF
END_FOR
IF T3S2sumavg > 0 THEN
	T3S2avg:=(T3S2sumavg/T3S2cnt3);	
END_IF	
T3.S2_fb(
	lettura:= REAL_TO_INT(T3S2avg), 
	maxScaleBit:= 32767, 
	maxScaleIng:= 1300, 
	deltaLowLimit:= 30,
	distanzaAVuoto:=590,
	valSoglia:= sogliaT3S2, 
	filterTime:=2,
	full=> T3.S2_full,
	actualVal=> T3.S2_actVal);


	

//SILOS1	
//CODA CIRCOLARE VALORI SENSORE inbit
S1SO2tmravg(IN:=TRUE,PT:=T#200MS);
S1SO2maxCnt:= REAL_TO_INT(S1SO2maxTimeavg*1000/200);
IF S1SO2maxCnt > 99 THEN
	S1SO2maxCnt:=99;
END_IF
IF S1SO2tmravg.Q THEN
	S1SO2tmravg(IN:=FALSE);	
	//CONTATORE TEMPO MASSIMO CAMPIONATURA
	IF S1SO2cnt < S1SO2maxCnt-1 THEN
		S1SO2cnt:=S1SO2cnt+1;	
	ELSE
		S1SO2cnt:=0;
	END_IF
	//POPOLO ARRAY LETTURE SENSORE in bit			
	S1SO2arravg[S1SO2cnt]:= S1_SO2;
END_IF
//MEDIA VALORI inbit
S1SO2cnt3:=0;
S1SO2sumavg:=0;
FOR S1SO2cnt2:=1 TO S1SO2maxCnt-1 DO
	IF S1SO2arravg[S1SO2cnt2] > 0 THEN
		S1SO2sumavg:= S1SO2sumavg + S1SO2arravg[S1SO2cnt2];
		S1SO2cnt3:=S1SO2cnt3+1;
	END_IF
END_FOR
IF S1SO2sumavg > 0 THEN
	S1SO2avg:=(S1SO2sumavg/S1SO2cnt3);	
END_IF
(*
S1.SO2_fb(
	lettura:= REAL_TO_INT(S1SO2avg), 
	maxScaleBit:= 32767, 
	maxScaleIng:= 6000, 
	deltaLowLimit:= 30, 
	distanzaAVuoto:=3250,
	valSoglia:= sogliaS1SO2, 
	filterTime:=1,
	full=> SO2_full_curr, //S1.SO2_full,
	actualVal=>S1.SO2_actVal);
	
	
	tmrValidaSoglia_S02(IN:= SO2_full_curr, PT:=T#15S);
	IF tmrValidaSoglia_S02.Q THEN
		tmrValidaSoglia_S02(IN:= FALSE);
		S1.SO2_full:= TRUE;
	END_IF
	
	IF NOT SO2_full_curr THEN
		S1.SO2_full:= FALSE;
	END_IF
	*)
	
//sensore livello silos (sensore in basso)

tmrS1_T_Rit_Empty(IN:=S1_S1,PT:=T#15m);
	S1.SO2_full:= TRUE;//tmrS1_T_Rit_Empty.Q OR Forza_TT1S01_Full;
	
//x HMI
glo_ES_ActVal.S1_S02:=S1.SO2_actVal;
altMatS1SO2:= S1.SO2_fb.distanzaAVuoto - glo_ES_ActVal.S1_S02;		
IF altMatS1SO2 <0 THEN
	altMatS1SO2:=0;
END_IF			
	


//SILOS2
S2.S1_fb(
	lettura:= S2_S1, 
	maxScaleBit:= 32767, 
	maxScaleIng:= 6000, 
	deltaLowLimit:= 30, 
	distanzaAVuoto:=6000,
	valSoglia:= 2000, 
	full=> S2.S1_full,
	actualVal=>S2.S1_actVal);
END_ACTION

END_PROGRAM

(* stored: Version 1.1.0.1, ProductVersion 3.1.4022.12
   POU EVACUAZIONE_SCARTI: Id {e1e90f84-2da5-421e-ac38-8582f800e994}, SpecialFunc None
   Action act_ALARM: Id {5ded8dbe-8890-4ab2-a626-b7c56d7ddc25}
   Action act_AreaMac_AUTO: Id {4299c151-616b-42a7-806f-5a6703d8c57a}
   Action act_AreaMac_MAN: Id {bef5b37c-250d-481b-88f3-c81af9c4d0fa}
   Action act_AreaSilos: Id {fbbd07a1-ba70-47aa-afaa-1b6eeda18dc2}
   Action act_HMI: Id {96798d00-c201-4db6-89ef-c78d6fd7f48c}
   Action act_INIT: Id {580611ca-94a3-4bcb-8752-e13d8ff1ce45}
   Action act_INPUT: Id {9c994c28-22a6-4f62-a8c2-2a9862140083}
   Action act_Macinatore: Id {587ecde4-fc76-4b85-b7a1-c25e2716cfdf}
   Action act_OUTPUT: Id {6e350841-508c-4dfd-aeea-77afb98e80fc}
   Action act_Semafori: Id {0db9c996-8963-4ea6-9007-70f6a4a157fb}
   Action act_Sensori: Id {d689a64f-5d94-4c3a-aecf-b9256c3086c6} *)
